(* CODESYS project Johnson,Joachim Projectredovisning Fisrst.project

Project tree, tasks and I/O mapping:
  Device : CODESYS Control Win V3, 3S - Smart Software Solutions GmbH, order no. 305021, version 3.5.10.40
    application Application
      libraries: Standard, * (System)
      task MainTask (cyclic, interval t#20ms, priority 1) calls Main
      task ProductWaitAlarm (cyclic, interval t#20ms, priority 1) calls ProductNotOffloadedAlarm
      task LightTower (cyclic, interval t#20ms, priority 1) calls LightSignals
      task HMI (cyclic, interval t#20ms, priority 1) calls HMI, ALARMtranslator
      global variables GVL
      Symbols
      Programs/
        Alarms/
          program ProductNotOffloadedAlarm [ST]
          program ALARMtranslator [ST]
          program Conv1Timeout [ST]
          program Conv2Timeout [ST]
          program Conv3Cyl3Timeout [ST]
          program Conv4Cyl4Timeout [ST]
          program Conv5Cyl5Timeout [ST]
        ConveyorMovment/
          program MoveBoxToScanner [CFC]
          program MoveToConveyer5 [CFC]
          program MoveToConveyer4 [CFC]
          program MoveToConveyer3 [CFC]
          program FromEndOfCylToOffload5 [CFC]
          program FromEndOfCylToOffload3 [CFC]
          program FromEndOfCylToOffload4 [CFC]
          program StopAllConv [CFC]
        SettParameters/
          program SetDirParameter [ST]
          program ResetParameters [ST]
          program StartUppParameters [ST]
      ProgamStruktures/
        program Main [SFC]
        program LightSignals [ST]
        program HMI [ST]
*)

// Device/Application/GVL
{attribute 'qualified_only'}
VAR_GLOBAL
	MaskinState: INT; // State of the maskin. 1 automode. 2 idle 3 stopp.
	Size: WORD;
	AlarmCode: WORD; // 0 = no alarm
	alarmOrIdle: BOOL;
	GeneralTimeOutTime: TIME;
	
	// HMI
	iSUB000_S1: BOOL; // Start button
	iSUB000_S2: BOOL; // Stop button
	iSUB000_S3: BOOL; // Reset button
	
	oSUB000_H1: BOOL; // Start button lamp
	oSUB000_H2: WORD; // Display
	oSUB000_H3: BOOL; // Reset button lamp
	
	// Beacoon
	oSUB000_H4: BOOL; // Beacon Green
	oSUB000_H5: BOOL; // Beacon Yellow
	oSUB000_H6: BOOL; // Beacon Red
	
	// Sub 10 convayor
	iSUB010_B1: BOOL; // Early sensor
	iSUB010_B2: BOOL; // Lower Sensor
	iSUB010_B3: BOOL; // Mid Sensor
	iSUB010_B4: BOOL; // High sensor
	oSUB010_K1: BOOL; // Motor FWD
	
	// Sub 20 convayor
	iSUB020_B1: BOOL; // Early sensor
	iSUB020_B2: BOOL; // Mid sensor
	iSUB020_B3: BOOL; // Late sensor
	oSUB020_K1: BOOL; // Motor FWD
	
	// Sub 30 convayor
	iSUB030_B1: BOOL; // Early sensor
	iSUB030_B2: BOOL; // Late sensor
	oSUB030_K1: BOOL; // Motor FWD
	oSUB030_Y1: BOOL; // Cylinder Expand
	iSUB030_C1_B1: BOOL; // Cylinder Expanded Sensor
	
	// Sub 40 convayor
	iSUB040_B1: BOOL; // Early sensor
	iSUB040_B2: BOOL; // LateSensor
	oSUB040_K1: BOOL; // Motor FWD
	oSUB040_Y1: BOOL; // Cylinder Expand
	iSUB040_C1_B1: BOOL; // Cylinder Expanded Sensor
	
	// Sub 50 convayor
	iSUB050_B1: BOOL; // Early sensor
	iSUB050_B2: BOOL; // LateSensor
	oSUB050_K1: BOOL; // Motor FWD
	oSUB050_Y1: BOOL; // Cylinder Expand
	iSUB050_C1_B1: BOOL; // Cylinder Expanded Sensor
	
END_VAR

// Device/Application/ProgamStruktures/Main
PROGRAM Main
VAR
	Size: WORD;
END_VAR

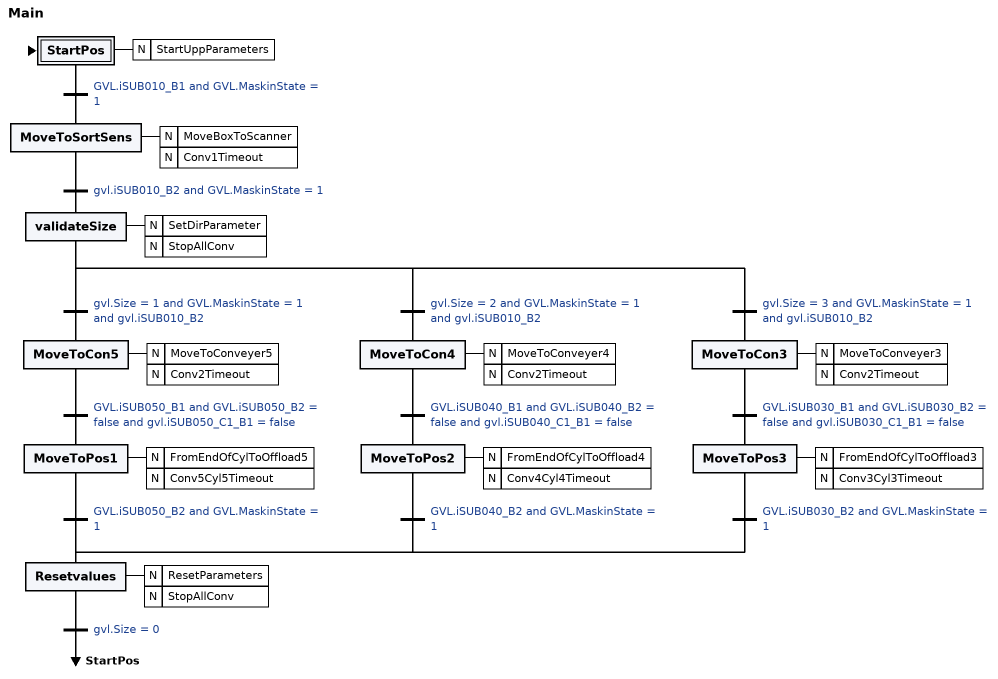
INITIAL_STEP StartPos:
    StartUppParameters(N);
END_STEP
TRANSITION FROM StartPos TO MoveToSortSens
    := GVL.iSUB010_B1 and GVL.MaskinState = 1;
END_TRANSITION
STEP MoveToSortSens:
    MoveBoxToScanner(N);
    Conv1Timeout(N);
END_STEP
TRANSITION FROM MoveToSortSens TO validateSize
    := gvl.iSUB010_B2 and GVL.MaskinState = 1;
END_TRANSITION
STEP validateSize:
    SetDirParameter(N);
    StopAllConv(N);
END_STEP
TRANSITION FROM validateSize TO MoveToCon5
    := gvl.Size = 1 and GVL.MaskinState = 1 and gvl.iSUB010_B2;
END_TRANSITION
STEP MoveToCon5:
    MoveToConveyer5(N);
    Conv2Timeout(N);
END_STEP
TRANSITION FROM MoveToCon5 TO MoveToPos1
    := GVL.iSUB050_B1 and GVL.iSUB050_B2 = false and gvl.iSUB050_C1_B1 = false;
END_TRANSITION
STEP MoveToPos1:
    FromEndOfCylToOffload5(N);
    Conv5Cyl5Timeout(N);
END_STEP
TRANSITION FROM MoveToPos1 TO Resetvalues
    := GVL.iSUB050_B2 and GVL.MaskinState = 1;
END_TRANSITION
TRANSITION FROM validateSize TO MoveToCon4
    := gvl.Size = 2 and GVL.MaskinState = 1 and gvl.iSUB010_B2;
END_TRANSITION
STEP MoveToCon4:
    MoveToConveyer4(N);
    Conv2Timeout(N);
END_STEP
TRANSITION FROM MoveToCon4 TO MoveToPos2
    := GVL.iSUB040_B1 and GVL.iSUB040_B2 = false and gvl.iSUB040_C1_B1 = false;
END_TRANSITION
STEP MoveToPos2:
    FromEndOfCylToOffload4(N);
    Conv4Cyl4Timeout(N);
END_STEP
TRANSITION FROM MoveToPos2 TO Resetvalues
    := GVL.iSUB040_B2 and GVL.MaskinState = 1;
END_TRANSITION
TRANSITION FROM validateSize TO MoveToCon3
    := gvl.Size = 3 and GVL.MaskinState = 1 and gvl.iSUB010_B2;
END_TRANSITION
STEP MoveToCon3:
    MoveToConveyer3(N);
    Conv2Timeout(N);
END_STEP
TRANSITION FROM MoveToCon3 TO MoveToPos3
    := GVL.iSUB030_B1 and GVL.iSUB030_B2 = false and gvl.iSUB030_C1_B1 = false;
END_TRANSITION
STEP MoveToPos3:
    FromEndOfCylToOffload3(N);
    Conv3Cyl3Timeout(N);
END_STEP
TRANSITION FROM MoveToPos3 TO Resetvalues
    := GVL.iSUB030_B2 and GVL.MaskinState = 1;
END_TRANSITION
STEP Resetvalues:
    ResetParameters(N);
    StopAllConv(N);
END_STEP
TRANSITION FROM Resetvalues TO StartPos
    := gvl.Size = 0;
END_TRANSITION

END_PROGRAM

// Device/Application/Programs/Alarms/ProductNotOffloadedAlarm
PROGRAM ProductNotOffloadedAlarm
VAR
	TimeOutAlarmcConv3: BOOL;
	TimeOutAlarmTimerConv3: Ton;
	
	TimeOutAlarmcConv4: BOOL;
	TimeOutAlarmTimerConv4: Ton;
	
	TimeOutAlarmcConv5: BOOL;
	TimeOutAlarmTimerConv5: Ton;
END_VAR

IF gvl.iSUB030_B2
	THEN
	TimeOutAlarmTimerConv3(IN:=gvl.oSUB030_K1, PT:=gvl.GeneralTimeOutTime);

	TimeOutAlarmcConv3 := TimeOutAlarmTimerConv3.q;
END_IF

IF gvl.iSUB040_B2
	THEN
	TimeOutAlarmTimerConv3(IN:=gvl.oSUB030_K1, PT:=gvl.GeneralTimeOutTime);

	TimeOutAlarmcConv3 := TimeOutAlarmTimerConv3.q;
END_IF

IF gvl.iSUB050_B2
	THEN
	TimeOutAlarmTimerConv3(IN:=gvl.oSUB030_K1, PT:=gvl.GeneralTimeOutTime);

	TimeOutAlarmcConv3 := TimeOutAlarmTimerConv3.q;
END_IF

// setting alarmcode for cylinder
IF TimeOutAlarmcConv3
	THEN
		gvl.MaskinState := 3;
		gvl.AlarmCode := 10;
END_IF

// setting alarmcode for cylinder
IF TimeOutAlarmcConv4
	THEN
		gvl.MaskinState := 3;
		gvl.AlarmCode := 10;
END_IF

// setting alarmcode for cylinder
IF TimeOutAlarmcConv5
	THEN
		gvl.MaskinState := 3;
		gvl.AlarmCode := 10; // 10 därför att larmet för gamla 10 tog bort på rekomendation.
END_IF

END_PROGRAM

// Device/Application/ProgamStruktures/LightSignals
PROGRAM LightSignals
VAR
END_VAR

IF GVL.MaskinState = 1
	THEN
		gvl.oSUB000_H4 := TRUE;
	ELSE
		gvl.oSUB000_H4 := FALSE;
END_IF

IF GVL.MaskinState = 2
	THEN
		gvl.oSUB000_H5 := TRUE;
	ELSE
		gvl.oSUB000_H5 := FALSE;
END_IF

IF GVL.MaskinState = 3
	THEN
		gvl.oSUB000_H6 := TRUE;
	ELSE
		gvl.oSUB000_H6 := FALSE;
END_IF

END_PROGRAM

// Device/Application/ProgamStruktures/HMI
PROGRAM HMI
VAR
	StarTimer: TON;
	TimeOutCounter: TIME;
END_VAR

// Button set maskinstate
IF GVL.iSUB000_S1 = TRUE AND gvl.MaskinState < 3
	THEN
		StarTimer(IN:=GVL.iSUB000_S1, PT:=gvl.GeneralTimeOutTime);
		gvl.MaskinState := 1;
END_IF

IF GVL.iSUB000_S2 = FALSE
	THEN
		gvl.MaskinState := 2;
END_IF

IF GVL.iSUB000_S3 = TRUE AND gvl.MaskinState = 3
	THEN
		gvl.MaskinState := 2;
		gvl.AlarmCode 	:= 0;
		GVL.alarmOrIdle := FALSE;
END_IF

// Printing out alarmcode. if 0 = no alarm
IF gvl.AlarmCode >= 0
	THEN
		gvl.oSUB000_H2 := gvl.AlarmCode;
END_IF

// Button Lights
IF GVL.MaskinState = 1
	THEN
		gvl.oSUB000_H1 := TRUE;
	ELSE
		gvl.oSUB000_H1 := FALSE;
END_IF

IF GVL.MaskinState = 3
	THEN
		gvl.oSUB000_H3 := TRUE;
	ELSE
		gvl.oSUB000_H3 := FALSE;
END_IF

END_PROGRAM

// Device/Application/Programs/Alarms/ALARMtranslator
PROGRAM ALARMtranslator
VAR
END_VAR

IF gvl.AlarmCode >= 2
	THEN
		gvl.alarmOrIdle := TRUE;
	ELSE
		gvl.alarmOrIdle := FALSE;
END_IF

END_PROGRAM

// Device/Application/Programs/ConveyorMovment/MoveBoxToScanner
PROGRAM MoveBoxToScanner
VAR
	RunMemory: SR;
END_VAR
VAR // added by the converter: edge detectors and wires of the graphical bodies
    _w1, _w4 : ANY;
    _w2, _w3, _w5 : BOOL;
END_VAR

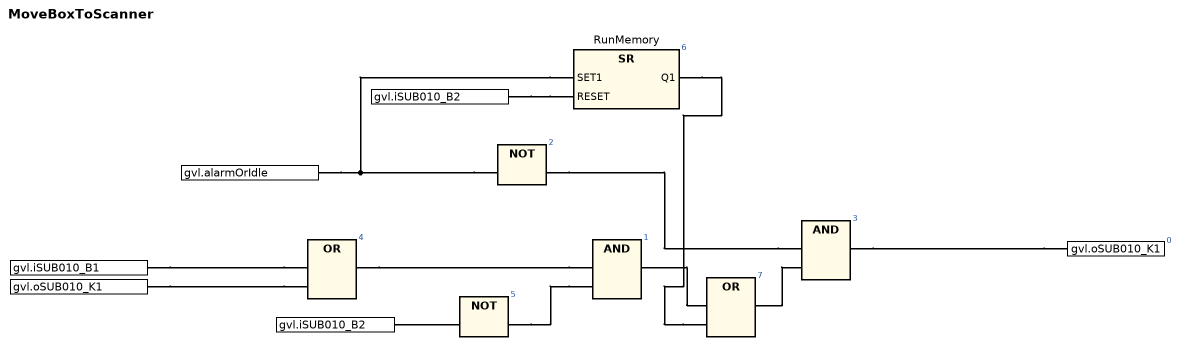
gvl.oSUB010_K1 := _w1;
_w4 := _w2 AND _w3;
_w1 := NOT gvl.alarmOrIdle AND _w5;
_w2 := gvl.iSUB010_B1 OR gvl.oSUB010_K1;
_w3 := NOT gvl.iSUB010_B2;
RunMemory(SET1 := gvl.alarmOrIdle, RESET := gvl.iSUB010_B2); // SR
_w5 := _w4 OR RunMemory.Q1;

END_PROGRAM

// Device/Application/Programs/SettParameters/SetDirParameter
PROGRAM SetDirParameter
VAR
END_VAR


IF gvl.iSUB010_B2
	THEN
		gvl.Size := 1;
END_IF
		
IF gvl.iSUB010_B3
	THEN
		gvl.Size := 2;
END_IF

IF gvl.iSUB010_B4
	THEN
		gvl.Size := 3;
END_IF

END_PROGRAM

// Device/Application/Programs/SettParameters/ResetParameters
PROGRAM ResetParameters
VAR
END_VAR

gvl.Size := 0;

END_PROGRAM

// Device/Application/Programs/ConveyorMovment/MoveToConveyer5
PROGRAM MoveToConveyer5
VAR
	RunMemory: SR;
	RunMemoryPush: SR;
END_VAR
VAR // added by the converter: edge detectors and wires of the graphical bodies
    _w1, _w4, _w6, _w7 : ANY;
    _w2, _w3, _w5, _w8 : BOOL;
END_VAR

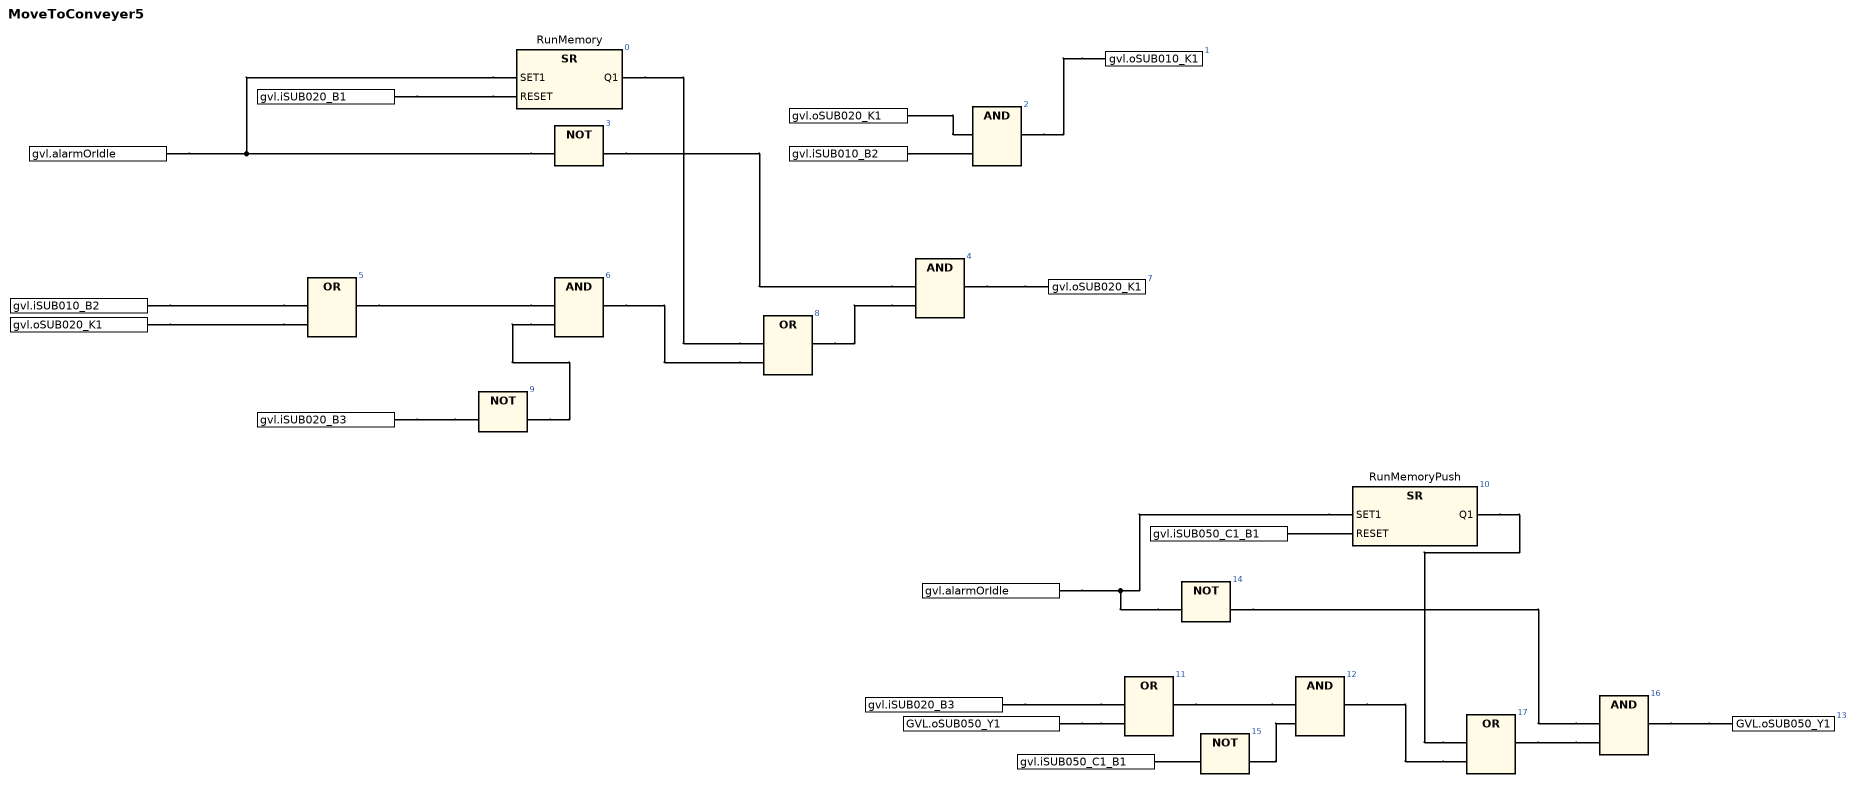
RunMemory(SET1 := gvl.alarmOrIdle, RESET := gvl.iSUB020_B1); // SR
gvl.oSUB010_K1 := _w1;
_w1 := gvl.oSUB020_K1 AND gvl.iSUB010_B2;
_w4 := (gvl.iSUB010_B2 OR gvl.oSUB020_K1) AND _w3;
gvl.oSUB020_K1 := NOT gvl.alarmOrIdle AND _w2;
_w2 := RunMemory.Q1 OR _w4;
_w3 := NOT gvl.iSUB020_B3;
RunMemoryPush(SET1 := gvl.alarmOrIdle, RESET := gvl.iSUB050_C1_B1); // SR
_w6 := (gvl.iSUB020_B3 OR GVL.oSUB050_Y1) AND _w5;
GVL.oSUB050_Y1 := _w7;
_w5 := NOT gvl.iSUB050_C1_B1;
_w7 := NOT gvl.alarmOrIdle AND _w8;
_w8 := RunMemoryPush.Q1 OR _w6;

END_PROGRAM

// Device/Application/Programs/ConveyorMovment/MoveToConveyer4
PROGRAM MoveToConveyer4
VAR
	RunMemory: SR;
	RunMemoryPush: SR;
END_VAR
VAR // added by the converter: edge detectors and wires of the graphical bodies
    _w1, _w3, _w5, _w7, _w8 : ANY;
    _w2, _w4, _w6, _w9 : BOOL;
END_VAR

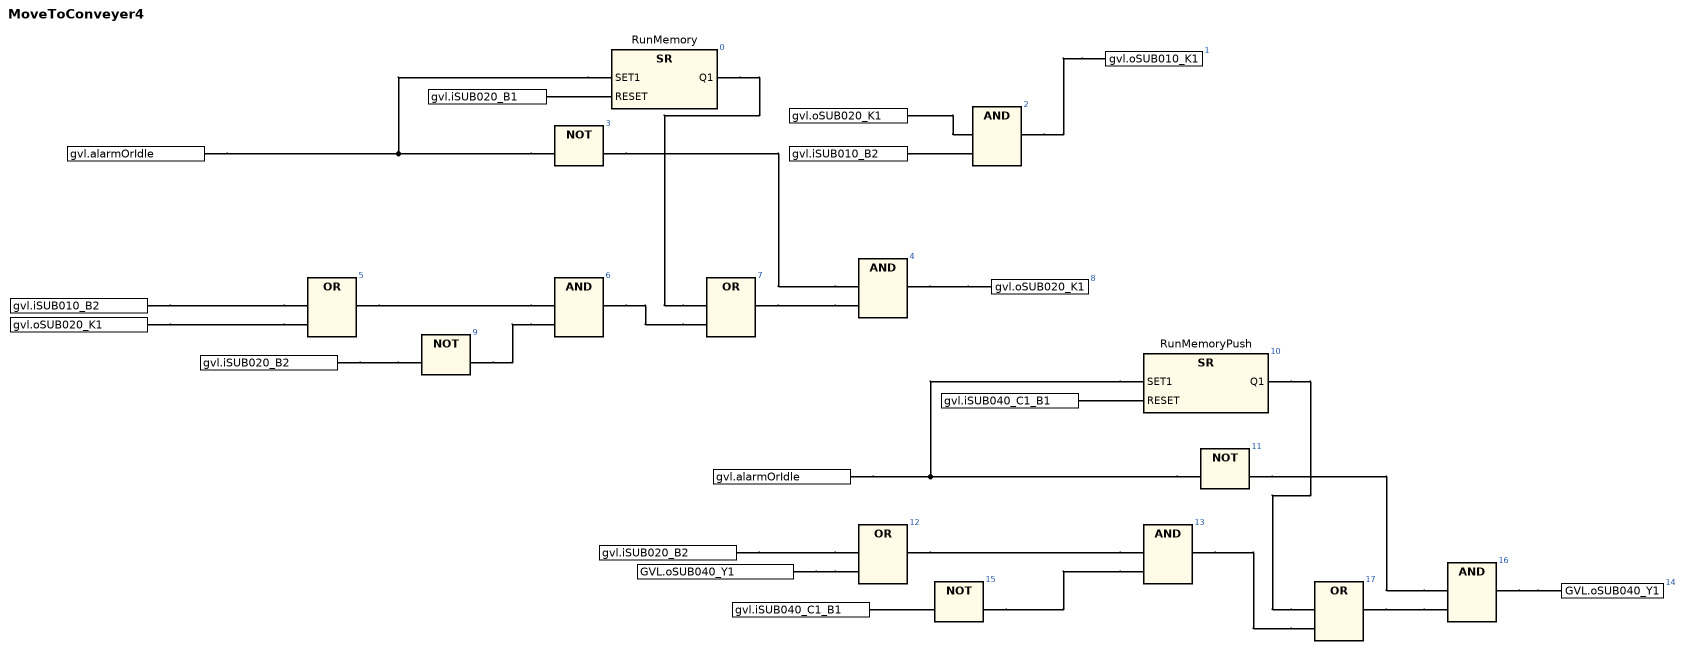
RunMemory(SET1 := gvl.alarmOrIdle, RESET := gvl.iSUB020_B1); // SR
gvl.oSUB010_K1 := _w1;
_w1 := gvl.oSUB020_K1 AND gvl.iSUB010_B2;
_w3 := NOT gvl.alarmOrIdle AND _w2;
_w2 := RunMemory.Q1 OR (gvl.iSUB010_B2 OR gvl.oSUB020_K1) AND _w4;
gvl.oSUB020_K1 := _w3;
_w4 := NOT gvl.iSUB020_B2;
RunMemoryPush(SET1 := gvl.alarmOrIdle, RESET := gvl.iSUB040_C1_B1); // SR
_w5 := NOT gvl.alarmOrIdle;
_w7 := (gvl.iSUB020_B2 OR GVL.oSUB040_Y1) AND _w6;
GVL.oSUB040_Y1 := _w8;
_w6 := NOT gvl.iSUB040_C1_B1;
_w8 := _w5 AND _w9;
_w9 := RunMemoryPush.Q1 OR _w7;

END_PROGRAM

// Device/Application/Programs/ConveyorMovment/MoveToConveyer3
PROGRAM MoveToConveyer3
VAR
	RunMemorys: SR;
	RunMemoryPusher: SR;
END_VAR
VAR // added by the converter: edge detectors and wires of the graphical bodies
    _w1, _w2, _w3, _w4, _w6, _w9 : ANY;
    _w5, _w7, _w8, _w10 : BOOL;
END_VAR

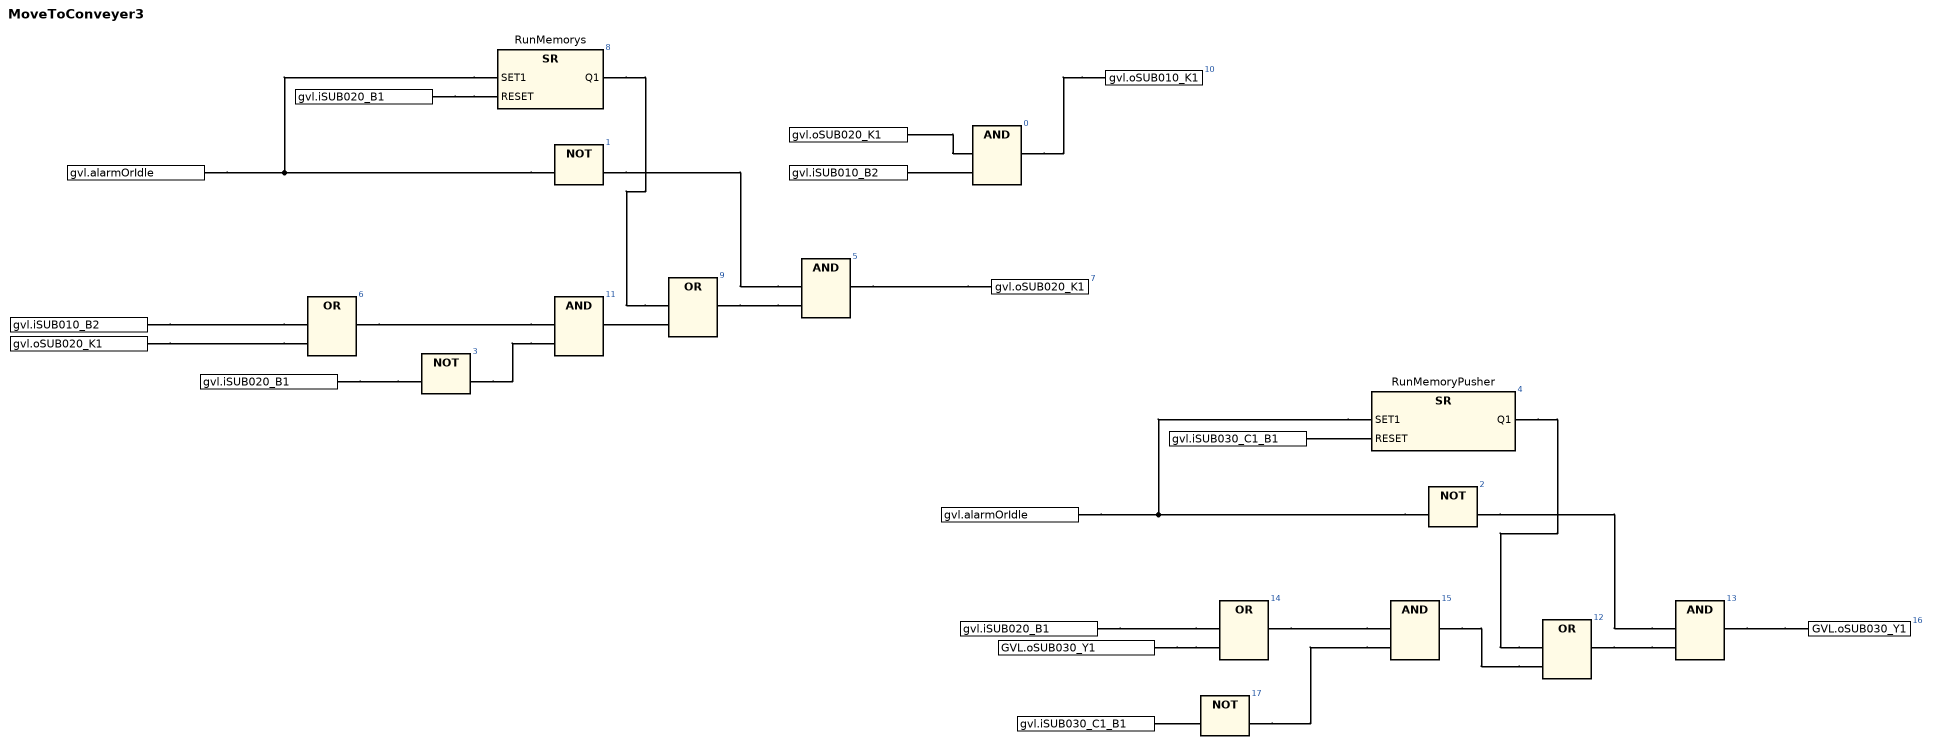
// note: 4 stored wires end on pins the file does not list and are not shown
_w1 := gvl.oSUB020_K1 AND gvl.iSUB010_B2;
_w2 := NOT gvl.alarmOrIdle;
_w3 := NOT gvl.alarmOrIdle;
_w4 := NOT gvl.iSUB020_B1;
RunMemoryPusher(SET1 := gvl.alarmOrIdle, RESET := gvl.iSUB030_C1_B1); // SR
_w6 := gvl.iSUB010_B2 OR gvl.oSUB020_K1;
gvl.oSUB020_K1 := _w2 AND _w5;
RunMemorys(SET1 := gvl.alarmOrIdle, RESET := gvl.iSUB020_B1); // SR
_w5 := RunMemorys.Q1 OR _w7;
gvl.oSUB010_K1 := _w1;
_w7 := _w6 AND _w4;
_w9 := _w3 AND (RunMemoryPusher.Q1 OR _w8);
_w8 := (gvl.iSUB020_B1 OR GVL.oSUB030_Y1) AND _w10;
GVL.oSUB030_Y1 := _w9;
_w10 := NOT gvl.iSUB030_C1_B1;

END_PROGRAM

// Device/Application/Programs/ConveyorMovment/FromEndOfCylToOffload5
PROGRAM FromEndOfCylToOffload5
VAR
	RunMemory: SR;
END_VAR
VAR // added by the converter: edge detectors and wires of the graphical bodies
    _w1, _w3 : BOOL;
    _w2 : ANY;
END_VAR

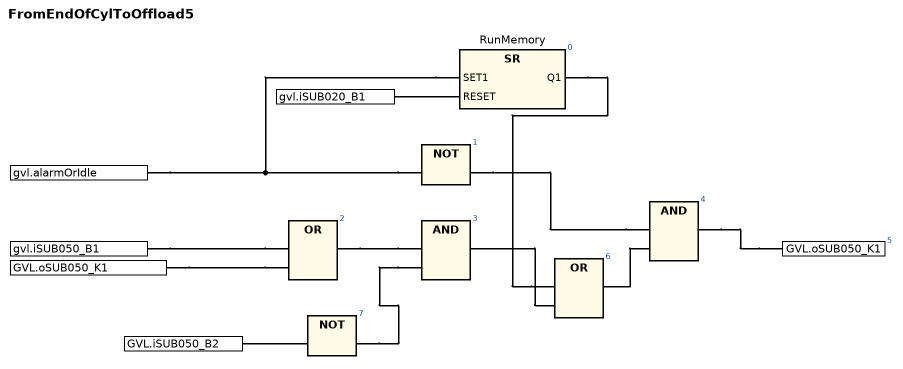
RunMemory(SET1 := gvl.alarmOrIdle, RESET := gvl.iSUB020_B1); // SR
_w2 := (gvl.iSUB050_B1 OR GVL.oSUB050_K1) AND _w1;
GVL.oSUB050_K1 := NOT gvl.alarmOrIdle AND _w3;
_w3 := RunMemory.Q1 OR _w2;
_w1 := NOT GVL.iSUB050_B2;

END_PROGRAM

// Device/Application/Programs/ConveyorMovment/FromEndOfCylToOffload3
PROGRAM FromEndOfCylToOffload3
VAR
	RunMemory: SR;
END_VAR
VAR // added by the converter: edge detectors and wires of the graphical bodies
    _w1, _w3, _w4 : ANY;
    _w2, _w5 : BOOL;
END_VAR

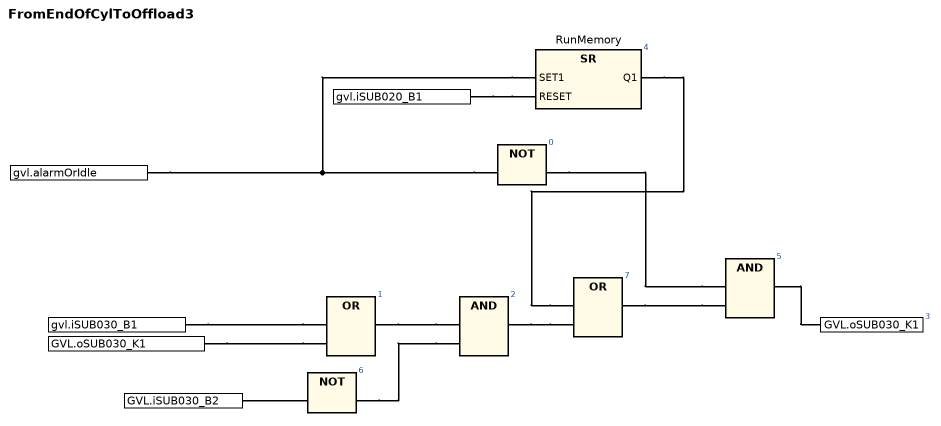
_w1 := NOT gvl.alarmOrIdle;
_w3 := (gvl.iSUB030_B1 OR GVL.oSUB030_K1) AND _w2;
GVL.oSUB030_K1 := _w4;
RunMemory(SET1 := gvl.alarmOrIdle, RESET := gvl.iSUB020_B1); // SR
_w4 := _w1 AND _w5;
_w2 := NOT GVL.iSUB030_B2;
_w5 := RunMemory.Q1 OR _w3;

END_PROGRAM

// Device/Application/Programs/ConveyorMovment/FromEndOfCylToOffload4
PROGRAM FromEndOfCylToOffload4
VAR
	RunMemorys: SR;
END_VAR
VAR // added by the converter: edge detectors and wires of the graphical bodies
    _w1, _w3 : BOOL;
    _w2 : ANY;
END_VAR

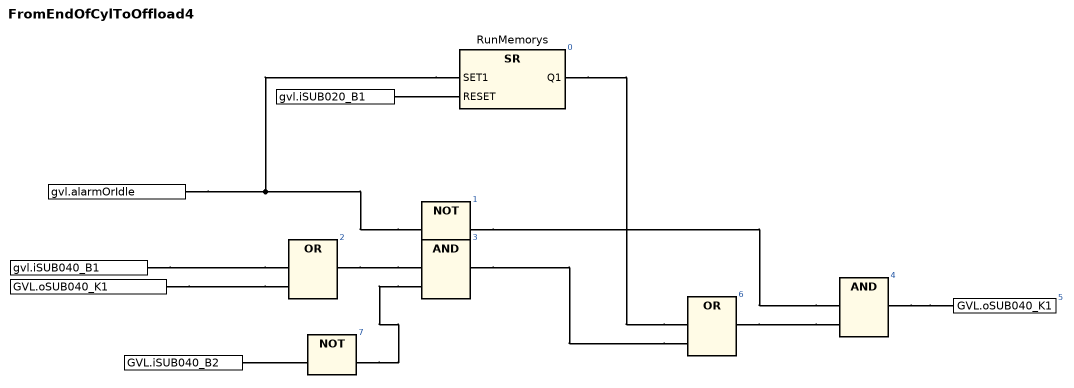
RunMemorys(SET1 := gvl.alarmOrIdle, RESET := gvl.iSUB020_B1); // SR
_w2 := (gvl.iSUB040_B1 OR GVL.oSUB040_K1) AND _w1;
GVL.oSUB040_K1 := NOT gvl.alarmOrIdle AND _w3;
_w3 := RunMemorys.Q1 OR _w2;
_w1 := NOT GVL.iSUB040_B2;

END_PROGRAM

// Device/Application/Programs/ConveyorMovment/StopAllConv
PROGRAM StopAllConv
VAR
END_VAR

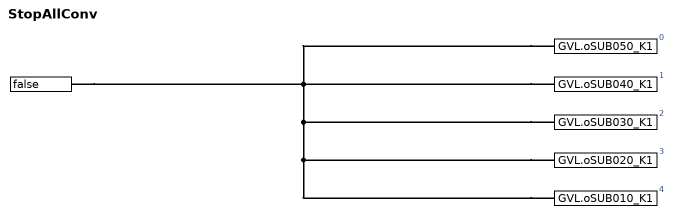
GVL.oSUB050_K1 := false;
GVL.oSUB040_K1 := false;
GVL.oSUB030_K1 := false;
GVL.oSUB020_K1 := false;
GVL.oSUB010_K1 := false;

END_PROGRAM

// Device/Application/Programs/SettParameters/StartUppParameters
PROGRAM StartUppParameters
VAR
END_VAR

// Setting up some standard values of alarms.
GVL.GeneralTimeOutTime := T#15S;

END_PROGRAM

// Device/Application/Programs/Alarms/Conv1Timeout
PROGRAM Conv1Timeout
VAR
	TimeOutAlarm: BOOL;
	TimeOutAlarmTimer: TON;
	TimeOutCounter: TIME;
END_VAR

TimeOutAlarmTimer(IN:=gvl.oSUB010_K1, PT:=gvl.GeneralTimeOutTime);

TimeOutAlarm := TimeOutAlarmTimer.q;

IF TimeOutAlarm
	THEN
		gvl.MaskinState := 3;
		gvl.AlarmCode := 1;
END_IF

END_PROGRAM

// Device/Application/Programs/Alarms/Conv2Timeout
PROGRAM Conv2Timeout
VAR
	TimeOutAlarm: BOOL;
	TimeOutAlarmTimer: TON;
	TimeOutCounter: TIME;
END_VAR

TimeOutAlarmTimer(IN:=gvl.oSUB020_K1, PT:=gvl.GeneralTimeOutTime);

TimeOutAlarm := TimeOutAlarmTimer.q;

IF TimeOutAlarm
	THEN
		gvl.MaskinState := 3;
		gvl.AlarmCode := 2;
END_IF

END_PROGRAM

// Device/Application/Programs/Alarms/Conv3Cyl3Timeout
PROGRAM Conv3Cyl3Timeout
VAR
	TimeOutAlarmCyl: BOOL;
	TimeOutAlarmcConvey: BOOL;
	TimeOutAlarmTimerConveyor: Ton;
	TimeOutAlarmTimerCylinder: Ton;
END_VAR

// Blev samma del av systemet med cylinder och tillhörande band. Får nämna i kommentarena om du tycker det ska delas.
IF gvl.iSUB050_B1
	THEN
	TimeOutAlarmTimerConveyor(IN:=gvl.oSUB030_K1, PT:=gvl.GeneralTimeOutTime);

	TimeOutAlarmcConvey := TimeOutAlarmTimerConveyor.q;
END_IF

IF gvl.oSUB030_Y1
	THEN
	TimeOutAlarmTimerCylinder(in:=gvl.iSUB020_B1, PT:=gvl.GeneralTimeOutTime);

	TimeOutAlarmCyl := TimeOutAlarmTimerCylinder.q;
END_IF

// setting alarmcode for convey
IF TimeOutAlarmcConvey
	THEN
		gvl.MaskinState := 3;
		gvl.AlarmCode := 3;
END_IF

// setting alarmcode for cylinder
IF TimeOutAlarmCyl
	THEN
		gvl.MaskinState := 3;
		gvl.AlarmCode := 6;
END_IF

END_PROGRAM

// Device/Application/Programs/Alarms/Conv4Cyl4Timeout
PROGRAM Conv4Cyl4Timeout
VAR
	TimeOutAlarmCyl: BOOL;
	TimeOutAlarmcConvey: BOOL;
	TimeOutAlarmTimerConveyor: Ton;
	TimeOutAlarmTimerCylinder: Ton;
END_VAR

// Blev samma del av systemet med cylinder och tillhörande band. Får nämna i kommentarena om du tycker det ska delas.
IF gvl.iSUB040_B1
	THEN
	TimeOutAlarmTimerConveyor(IN:=gvl.oSUB040_K1, PT:=gvl.GeneralTimeOutTime);

	TimeOutAlarmcConvey := TimeOutAlarmTimerConveyor.q;
END_IF

IF gvl.oSUB040_Y1
	THEN
	TimeOutAlarmTimerCylinder(in:=GVL.iSUB020_B2, PT:=gvl.GeneralTimeOutTime);

	TimeOutAlarmCyl := TimeOutAlarmTimerCylinder.q;
END_IF

// setting alarmcode for convey
IF TimeOutAlarmcConvey
	THEN
		gvl.MaskinState := 3;
		gvl.AlarmCode := 4;
END_IF

// setting alarmcode for cylinder
IF TimeOutAlarmCyl
	THEN
		gvl.MaskinState := 3;
		gvl.AlarmCode := 7;
END_IF

END_PROGRAM

// Device/Application/Programs/Alarms/Conv5Cyl5Timeout
PROGRAM Conv5Cyl5Timeout
VAR
	TimeOutAlarmCyl: BOOL;
	TimeOutAlarmcConvey: BOOL;
	TimeOutAlarmTimerConveyor: TON;
	TimeOutAlarmTimerCylinder: Ton;
END_VAR

// Blev samma del av systemet med cylinder och tillhörande band. Får nämna i kommentarena om du tycker det ska delas.
IF gvl.iSUB050_B1
	THEN
	TimeOutAlarmTimerConveyor(IN:=gvl.oSUB050_K1, PT:=gvl.GeneralTimeOutTime);

	TimeOutAlarmcConvey := TimeOutAlarmTimerConveyor.q;
END_IF

IF gvl.oSUB030_Y1
	THEN
	TimeOutAlarmTimerCylinder(in:=GVL.iSUB020_B3, PT:=gvl.GeneralTimeOutTime);

	TimeOutAlarmCyl := TimeOutAlarmTimerCylinder.q;
END_IF

// setting alarmcode for convey
IF TimeOutAlarmcConvey
	THEN
		gvl.MaskinState := 3;
		gvl.AlarmCode := 5;
END_IF

// setting alarmcode for cylinder
IF TimeOutAlarmCyl
	THEN
		gvl.MaskinState := 3;
		gvl.AlarmCode := 8;
END_IF

END_PROGRAM
